FUNCTION_BLOCK FB_DCAxis
VAR_INPUT
	open,
	close,
	enable,
	reset,
	limit_open,
	limit_close: 		BOOL;
	velocity:			INT := 24000;
	Threshold_active:	BOOL;
END_VAR
VAR_OUTPUT
	error,
	warning: BOOL;
	Ready_to_enable:	BOOL;
	Ready:				BOOL;
	Moving_negative:	BOOL;
	Moving_positive:	BOOL;
	Digital_input1:		BOOL;
	Digital_input2:		BOOL;
END_VAR
VAR_IN_OUT
	axis_ref:	MDP5001_511_733_FFF278FE;
END_VAR
VAR
	enable_state: RS;
END_VAR

enable_state(SET := enable AND Ready_to_enable,
			 RESET1 := reset);			
axis_ref.MDP5001_511_733_Output.MDP5001_733_Velocity := 0;
IF open AND limit_open THEN
	axis_ref.MDP5001_511_733_Output.MDP5001_733_Velocity := velocity;
END_IF

IF close AND limit_close THEN
	axis_ref.MDP5001_511_733_Output.MDP5001_733_Velocity := -velocity;
END_IF
axis_ref.MDP5001_511_733_Output.MDP5001_733_Control_1.Enable := enable_state.Q1;
axis_ref.MDP5001_511_733_Output.MDP5001_733_Control_1.Reset := reset;
axis_ref.MDP5001_511_733_Output.MDP5001_733_Control_1.Threshold_active := Threshold_active;

error := 	axis_ref.MDP5001_511_733_Input.MDP5001_733_Status_1.Error OR
			axis_ref.MDP5001_511_733_Input.MDP5001_733_Status_1.Sync_error;
			//(limit_open AND limit_close);
			//(open AND NOT limit_open) OR
			//(close AND NOT limit_close);
			
warning := axis_ref.MDP5001_511_733_Input.MDP5001_733_Status_1.Warning;

Ready_to_enable := axis_ref.MDP5001_511_733_Input.MDP5001_733_Status_1.Ready_to_enable;
Ready := axis_ref.MDP5001_511_733_Input.MDP5001_733_Status_1.Ready;

Moving_negative := axis_ref.MDP5001_511_733_Input.MDP5001_733_Status_1.Moving_negative;
Moving_positive := axis_ref.MDP5001_511_733_Input.MDP5001_733_Status_1.Moving_positive;

Digital_input1 := axis_ref.MDP5001_511_733_Input.MDP5001_733_Status_1.Digital_input_1;
Digital_input2 := axis_ref.MDP5001_511_733_Input.MDP5001_733_Status_1.Digital_input_2;

END_FUNCTION_BLOCK

(* stored: Version 1.1.0.1, ProductVersion 3.1.4024.12
   POU FB_DCAxis: Id {806daa9e-d8f7-460b-a5e1-6dcf9a5d40c4}, SpecialFunc None *)
